TYPE E_EcCommState : (
    eEcState_UNDEFINED 	:= 0,
    eEcState_INIT 		:= 1,
    eEcState_PREOP 		:= 2,
    eEcState_BOOT 		:= 3,
    eEcState_SAFEOP 	:= 4,
    eEcState_OP 		:= 8
) UDINT;
END_TYPE

(* stored: Version 1.1.0.1, ProductVersion 3.1.4022.18
   DUT E_EcCommState: Id {4385ddb9-c8b3-4c31-9540-480380e7b3e2} *)
